# EPICS autosave request: iocBoot/ioc13MCC/auto_positions.req
file "CARS_motor_positions.req",         P=$(P), M=m1
file "CARS_motor_positions.req",         P=$(P), M=m2
file "CARS_motor_positions.req",         P=$(P), M=m3
